Yaskawa INFORM job: TESTADRIAN.JBI

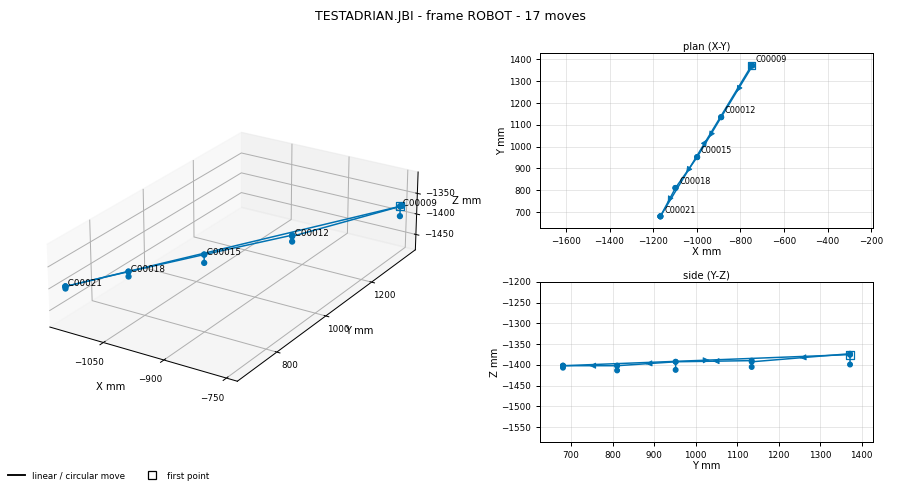
[picture p0: tool path of TESTADRIAN.JBI in frame ROBOT, 17 of 32 moves have a stored position in this frame; points joined in program order, loops and branches not executed]
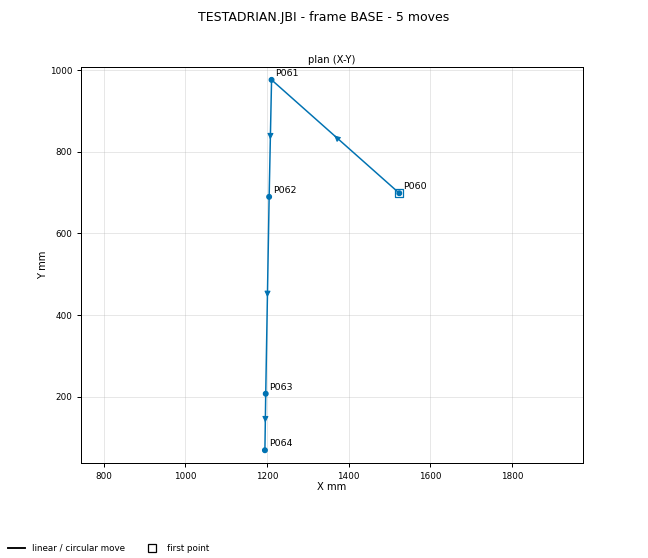
[picture p1: tool path of TESTADRIAN.JBI in frame BASE, 5 of 32 moves have a stored position in this frame; points joined in program order, loops and branches not executed]
/JOB
//NAME TESTADRIAN
//POS
///NPOS 26,26,0,11,0,0
///TOOL 0
///POSTYPE ROBOT
///RECTAN
///RCONF 0,0,0,0,0,0,0,0,0,0,0,0,0,0,0,0,0,0,0,0,0,0,0,0
C00000=-1035.526,919.929,-1397.692,9.2479,37.0905,-34.2442
C00001=-1033.556,915.270,-1401.300,9.2482,37.0867,-34.2473
C00002=-1055.783,915.269,-1401.301,9.2478,37.0866,-34.2497
C00003=-1033.563,915.268,-1411.965,9.2468,37.0870,-34.2499
C00004=-1035.526,919.929,-1397.692,9.2479,37.0905,-34.2442
C00005=-940.546,1065.827,-1396.144,9.2504,37.0853,-34.2465
C00006=-940.546,1065.827,-1396.144,9.2504,37.0853,-34.2465
C00007=-962.855,1065.824,-1396.160,9.2497,37.0848,-34.2481
C00008=-940.539,1065.834,-1408.722,9.2506,37.0852,-34.2483
C00009=-749.229,1371.947,-1375.142,19.2122,25.3194,54.7649
C00010=-749.245,1371.950,-1399.047,19.2137,25.3200,54.7650
C00011=-744.062,1371.872,-1373.000,19.2081,25.3216,54.7703
C00012=-888.177,1135.095,-1392.458,19.2114,25.3213,54.7713
C00013=-888.162,1135.097,-1404.947,19.2099,25.3206,54.7706
C00014=-888.146,1135.084,-1389.652,19.2087,25.3204,54.7704
C00015=-998.229,951.939,-1392.438,19.2128,25.3209,54.7710
C00016=-998.233,951.922,-1411.952,19.2120,25.3232,54.7675
C00017=-998.229,951.939,-1392.438,19.2128,25.3209,54.7710
C00018=-1097.615,810.935,-1401.902,19.2120,25.3247,54.7673
C00019=-1097.623,810.930,-1413.261,19.2123,25.3249,54.7692
C00020=-1097.615,810.935,-1401.902,19.2120,25.3247,54.7673
C00021=-1166.866,680.528,-1401.915,19.2113,25.3228,54.7692
C00022=-1166.853,680.530,-1406.722,19.2105,25.3220,54.7693
C00023=-1166.866,680.528,-1401.915,19.2113,25.3228,54.7692
C00024=-749.229,1371.947,-1375.142,19.2122,25.3194,54.7649
C00025=-1166.866,680.528,-1401.915,19.2113,25.3228,54.7692
BC00000=1602.617,32.863,1148.397
BC00001=1602.617,32.863,1148.397
BC00002=1602.617,32.863,1148.397
BC00003=1602.617,32.863,1148.397
BC00004=1602.617,32.863,1148.397
BC00005=1602.617,32.863,1148.397
BC00006=1602.617,32.863,1148.397
BC00007=1602.617,32.863,1148.397
BC00008=1602.617,32.863,1148.397
BC00009=1602.629,32.850,1148.408
BC00010=1602.629,32.850,1148.408
BC00011=1602.629,32.850,1148.408
BC00012=1602.629,32.850,1148.408
BC00013=1602.629,32.850,1148.408
BC00014=1602.629,32.850,1148.408
BC00015=1602.629,32.850,1148.408
BC00016=1602.629,32.850,1148.408
BC00017=1602.629,32.850,1148.408
BC00018=1602.629,32.850,1148.408
BC00019=1602.629,32.850,1148.408
BC00020=1602.629,32.850,1148.408
BC00021=1602.629,32.850,1148.408
BC00022=1602.629,32.850,1148.408
BC00023=1602.629,32.850,1148.408
BC00024=1602.629,32.850,1148.408
BC00025=1602.629,32.850,1148.408
///POSTYPE BASE
///RCONF 0,0,0,0,1,0,0,0,0,0,0,0,0,0,0,0,0,0,0,0,0,0,0,0
P00006=2.006,1.622,-0.565,0.0000,0.0000,0.0000
P00022=2.006,1.622,-0.565,0.0000,0.0000,0.0000
///RCONF 0,0,0,0,0,0,0,0,0,0,0,0,0,0,0,0,0,0,0,0,0,0,0,0
P00032=-0.423,0.157,3.222,0.0000,0.0000,0.0000
P00060=1524.284,698.404,-261.973,-0.4635,36.8346,-1.2388
P00061=1211.499,975.999,-261.374,0.5148,35.2356,175.5099
P00062=1205.574,689.500,-262.704,0.5159,35.2461,175.5270
P00063=1197.217,207.358,-268.729,0.4863,35.2395,175.4586
P00064=1195.199,68.975,-269.171,0.5092,35.2366,175.4908
P00099=-10.497,4.418,3.734,0.0000,0.0000,0.0000
P00125=0.000,0.000,2.400,0.0000,0.0000,0.0000
P00126=-50.000,0.000,0.000,0.0000,0.0000,0.0000
//INST
///DATE 2023/12/19 19:49
///ATTR SC,RW,RJ
////FRAME ROBOT
///GROUP1 RB1,BS1
NOP
COMM MOVJ C00000 BC00000 VJ=0.78
COMM REFP 3 C00001 BC00001
COMM REFP 4 C00002 BC00002
COMM REFP 5 C00003 BC00003
COMM CALL JOB:SEARCH
COMM SET P022 P006
COMM SETE P032 (3) D050
COMM SFTOF
COMM MOVL C00004 BC00004 V=16.7
COMM MOVL C00005 BC00005 V=16.7
COMM REFP 3 C00006 BC00006
COMM REFP 4 C00007 BC00007
COMM REFP 5 C00008 BC00008
COMM CALL JOB:SEARCH
COMM SET P022 P006
'1
MOVL C00009 BC00009 V=16.7
MOVL C00010 BC00010 V=16.7 SRCH RIN#(1)=ON T=1.00 DIS=20.0
IMOV P125 V=23.0
IMOV P126 V=23.0 SRCH RIN#(1)=ON DIS=20.0
TIMER T=0.10
GETS PX060 $PX001
TIMER T=0.10
MOVJ C00011 BC00011 VJ=0.78
'2
MOVL C00012 BC00012 V=50.0
MOVL C00013 BC00013 V=16.7 SRCH RIN#(1)=ON T=1.00 DIS=20.0
IMOV P125 V=23.0
IMOV P126 V=23.0 SRCH RIN#(1)=ON DIS=20.0
TIMER T=0.10
GETS PX061 $PX001
TIMER T=0.10
MOVJ C00014 BC00014 VJ=0.78
'3
MOVL C00015 BC00015 V=50.0
MOVL C00016 BC00016 V=16.7 SRCH RIN#(1)=ON T=1.00 DIS=20.0
IMOV P125 V=23.0
IMOV P126 V=23.0 SRCH RIN#(1)=ON DIS=20.0
TIMER T=0.10
GETS PX062 $PX001
TIMER T=0.10
MOVJ C00017 BC00017 VJ=0.78
'4
MOVL C00018 BC00018 V=50.0
MOVL C00019 BC00019 V=16.7 SRCH RIN#(1)=ON T=1.00 DIS=20.0
IMOV P125 V=23.0
IMOV P126 V=23.0 SRCH RIN#(1)=ON DIS=20.0
TIMER T=0.10
GETS PX063 $PX001
TIMER T=0.10
MOVJ C00020 BC00020 VJ=0.78
'5
MOVL C00021 BC00021 V=50.0
MOVL C00022 BC00022 V=16.7 SRCH RIN#(1)=ON T=1.00 DIS=20.0
IMOV P125 V=23.0
IMOV P126 V=23.0 SRCH RIN#(1)=ON DIS=20.0
TIMER T=0.10
GETS PX064 $PX001
TIMER T=0.10
MOVJ C00023 BC00023 VJ=0.78
'********
'********
'********
SFTON P099
MOVL C00024 BC00024 V=100.0
ARCON
MOVL P060 V=23.0
MOVL P061 V=23.0
MOVL P062 V=23.0
MOVL P063 V=23.0
MOVL P064 V=23.0
ARCOF
MOVJ C00025 BC00025 VJ=15.00
END
